PROGRAM PRG_12_OilContaminationAnalytics
VAR
	OilDiffPressSensor: GenericSensor;
	
	{attribute 'OPC.UA.DA' := '1'}
	{attribute 'OPC.UA.DA.Access' := '1'}			// read only
	{attribute 'OPC.UA.DA.StructuredType' := '1'}
	OilDiffPressSensorStruct			: SingleSensor_DataModel;
END_VAR

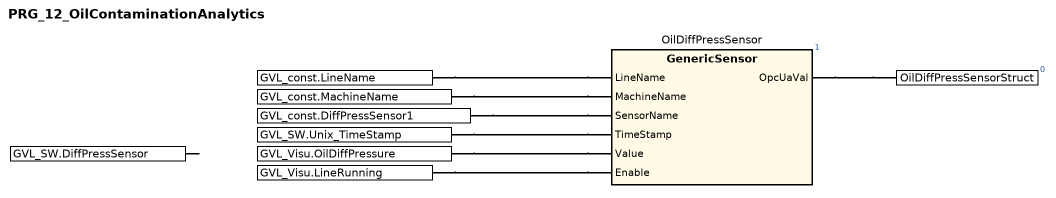
OilDiffPressSensorStruct := OilDiffPressSensor.OpcUaVal;
OilDiffPressSensor(
    LineName := GVL_const.LineName,
    MachineName := GVL_const.MachineName,
    SensorName := GVL_const.DiffPressSensor1,
    TimeStamp := GVL_SW.Unix_TimeStamp,
    Value := GVL_Visu.OilDiffPressure,
    Enable := GVL_Visu.LineRunning); // GenericSensor
// GVL_SW.DiffPressSensor: input not connected

END_PROGRAM

(* stored: Version 1.1.0.1, ProductVersion 3.1.4024.15
   POU PRG_12_OilContaminationAnalytics: Id {9509c8f2-193f-4e3b-9287-dc1013adfb72}, SpecialFunc None *)
